(* IEC 61131-3 sources: amr-agent/beckhoff/plc, 3 files *)

(* ---- GVL_IO.st ---- *)
// GVL_IO - the port of the m5_ver2 tag table (m5_ver2/CLAUDE.md section 3.1).
// One global variable list, written over ADS by exactly one process
// (beckhoff/windows/step5_tc.py) - the single-writer rule carries over.
//
// NAME MAPPING, the only one in the port: ST identifiers cannot carry a
// hyphen, so the Siemens tag `E-Stop` is `EStop` here. The UDP wire keys
// toward WSL are byte-identical to the m5_ver2 wire; the mapping lives in
// the writer's TAG table and nowhere else.
//
// Paste into: PLC project > GVLs > Add > Global Variable List, name GVL_IO.
{attribute 'qualified_only'}
VAR_GLOBAL
    // ---- written by the panel (the field devices' picture) ----
    EStop          : BOOL := FALSE;  // TRUE = healthy (NC chain closed)
    PF_OSSD        : BOOL := FALSE;  // TRUE = back protective field clear
    WF_Clear       : BOOL := FALSE;  // TRUE = back warning field clear
    PF_OSSD_right  : BOOL := FALSE;
    WF_Clear_right : BOOL := FALSE;
    PF_OSSD_left   : BOOL := FALSE;
    WF_Clear_left  : BOOL := FALSE;
    Acknowledge    : BOOL := FALSE;  // reset button, rising edge required
    ENC_A          : INT  := 0;      // encoder channel A, mm/s
    ENC_B          : INT  := 0;      // encoder channel B, mm/s

    // ---- computed by MAIN, read by the panel ----
    Motor          : BOOL := FALSE;  // the drive enable, AND of all chains
    CASE_B0        : BOOL := FALSE;  // monitoring-case bit 0
    CASE_B1        : BOOL := FALSE;  // monitoring-case bit 1
    V_Limit        : INT  := 300;    // speed ceiling mm/s; starts at creep -
                                     // not knowing is the slowest permission
END_VAR

(* ---- FB_ESTOP1.st ---- *)
// FB_ESTOP1 - the Siemens ESTOP1 semantics, ported to structured text.
//
// ROLE AND CLAIM, stated here because this file is where the logic lives:
// the safety chain is AUTHORED as a TE9000 safety project - the spec is
// beckhoff/plc/safety/SAFETY-APP.md - and this block is its STAND-IN
// EXECUTOR for the live loop until a safety runtime (TE9100 or TwinSAFE
// hardware) lands. It demonstrates the same observable semantics the
// F-block showed on PLCSIM Advanced; it carries NO safety integrity, no
// PL, Category, SIL or PFH (RESEARCH.md D3; ADR 0011 D5 discipline). The
// parity table (RUNBOOK part 5, S1-S6) pins it to the safety project.
//
// The semantics, measured on the F-CPU (m5_ver2/CLAUDE.md section 3.2):
//   - a demand LATCHES: the input returning to healthy does not re-enable
//   - clearing needs a RISING EDGE on Acknowledge, with the input healthy
//   - ACK_NEC: one Acknowledge is required after startup before Q can
//     ever be TRUE - hence demandLatched starts TRUE
//
// Paste into: PLC project > POUs > Add > POU, Function Block, ST.
FUNCTION_BLOCK FB_ESTOP1
VAR_INPUT
    S_In : BOOL;   // TRUE = healthy; FALSE = demand
    Ack  : BOOL;   // acknowledge button
END_VAR
VAR_OUTPUT
    Q : BOOL;      // enable: TRUE only with input healthy and no latch
END_VAR
VAR
    demandLatched : BOOL := TRUE;   // ACK_NEC: born latched, every startup
    ackPrev       : BOOL := TRUE;   // TRUE so a stuck-high Ack at startup
                                    // cannot count as an edge
END_VAR

IF NOT S_In THEN
    demandLatched := TRUE;                    // a demand latches
END_IF;
IF Ack AND NOT ackPrev AND S_In THEN
    demandLatched := FALSE;                   // rising edge, input healthy
END_IF;
ackPrev := Ack;
Q := S_In AND NOT demandLatched;

(* ---- MAIN.st ---- *)
// MAIN - the stand-in executor of the TE9000 safety application
// (beckhoff/plc/safety/SAFETY-APP.md), plus the standard-program half
// that TIA also kept standard: V_Limit and the case bits for the wire.
// When a safety runtime lands (TE9100 / TwinSAFE hardware), the five
// chains below reduce to mirroring the safety output into GVL_IO.Motor
// (RUNBOOK part 6); until then this file executes the chain live.
//
// Motor is the AND of five FB_ESTOP1 enables: e-stop button, three
// protective fields (back / right / left - the owner added right and left
// on 2026-08-12), and the speed monitor. WF_Clear is deliberately NOT in
// the Motor AND - measured on the F-CPU (step2/step3 PROOF: Motor TRUE
// with WF FALSE); it gates V_Limit, and through it the speed monitor.
//
// TWO TIA-SIDE BEHAVIOURS WERE NEVER MAPPED AND ARE PORTED CONSERVATIVELY,
// both labelled here and falling to the validation diff (RUNBOOK part 4):
//   - right/left warning-field composition into V_Limit (step5 PROOF open
//     item 4): ported as the conservative AND - ANY warning field occupied
//     drops the ceiling to 300.
//   - monitoring-case selection: ported as the constant case 1, the value
//     every live step5 run observed (case-1 fields 1.0 m / 2.5 m).
//
// Paste into: PLC project > POUs > MAIN (PRG), ST. Default PlcTask (10 ms).
PROGRAM MAIN
VAR
    chainEStop   : FB_ESTOP1;   // e-stop button
    chainPFBack  : FB_ESTOP1;   // back protective field
    chainPFRight : FB_ESTOP1;
    chainPFLeft  : FB_ESTOP1;
    chainSpeed   : FB_ESTOP1;   // encoder cross-check + ceilings
    speedHealthy : BOOL;
    diff         : INT;
    wfAllClear   : BOOL;
END_VAR

// V_Limit first: the speed monitor reads it this same cycle.
// 1500 with the warning fields clear, 300 otherwise - the measured law
// (step3 PROOF: creep demanded 0.68 s after enable near racking).
wfAllClear := GVL_IO.WF_Clear AND GVL_IO.WF_Clear_right
              AND GVL_IO.WF_Clear_left;
IF wfAllClear THEN
    GVL_IO.V_Limit := 1500;
ELSE
    GVL_IO.V_Limit := 300;
END_IF;

// The two-channel speed monitor, all three measured demands:
//   cross-check   |ENC_A - ENC_B| > 50 mm/s   (the fa/oa faults trip this)
//   ceiling       |ENC| > 2800 mm/s
//   case ceiling  |ENC| > V_Limit + 50        (the step3 creep trap)
// The +50 mm/s margin on the case ceiling is the PORT'S choice, labelled:
// the autopilot caps its command AT V_Limit, so the shaft rides exactly on
// the limit and a zero-margin compare would latch on measurement noise.
// The TIA implementation's own tolerance/delay was never mapped; this
// margin is the smallest that cannot chatter, and it falls to the
// validation diff like the other two unmapped behaviours.
diff := ABS(GVL_IO.ENC_A - GVL_IO.ENC_B);
speedHealthy := (diff <= 50)
    AND (ABS(GVL_IO.ENC_A) <= 2800) AND (ABS(GVL_IO.ENC_B) <= 2800)
    AND (ABS(GVL_IO.ENC_A) <= GVL_IO.V_Limit + 50)
    AND (ABS(GVL_IO.ENC_B) <= GVL_IO.V_Limit + 50);

// Five chains, one Acknowledge - the panel's RESET pulse clears them all,
// which is what the live F-CPU did too (measured 2026-08-13: a single
// Acknowledge cleared the right and left latches together).
chainEStop(S_In := GVL_IO.EStop, Ack := GVL_IO.Acknowledge);
chainPFBack(S_In := GVL_IO.PF_OSSD, Ack := GVL_IO.Acknowledge);
chainPFRight(S_In := GVL_IO.PF_OSSD_right, Ack := GVL_IO.Acknowledge);
chainPFLeft(S_In := GVL_IO.PF_OSSD_left, Ack := GVL_IO.Acknowledge);
chainSpeed(S_In := speedHealthy, Ack := GVL_IO.Acknowledge);

GVL_IO.Motor := chainEStop.Q AND chainPFBack.Q AND chainPFRight.Q
                AND chainPFLeft.Q AND chainSpeed.Q;

// Case bits: 01 = case 1, pinned (see the header). The vehicle's
// field_eval maps an unreadable 00 to case 3, the largest field - that
// fail direction lives on the consumer and is not re-implemented here.
GVL_IO.CASE_B0 := TRUE;
GVL_IO.CASE_B1 := FALSE;
